// TIA Portal V15 export
// export: Created 2018-05-29T12:25:38.1552518Z, ExportSetting WithDefaults, DisplayName Totally Integrated Automation Portal, DisplayVersion V15, DisplayName TIA Portal Openness, DisplayVersion V15, DisplayName STEP 7 Professional, DisplayVersion V15, DisplayName WinCC Professional, DisplayVersion V15
FUNCTION "Control_Modules" : Void   // FC1, STL
TITLE = Program
{ S7_Optimized_Access := 'TRUE' }
VERSION : 0.1
// Call all the Control Modules
// stored: AutoNumber true, UDAEnableTagReadback false
BEGIN

NETWORK
TITLE = Main
// comment
	CALL	XV001_fc
	CALL	XV002_fc
	CALL	XV003_fc
	CALL	XV004_fc
	CALL	XV300_fc
	CALL	XV400_fc
	CALL	XV500_fc
	CALL	XV301_fc
	CALL	XV501_fc
	CALL	XV401_fc
	CALL	MV001_fc
	CALL	MV002_fc
	CALL	MV003_fc
	CALL	MV004_fc
	CALL	MV005_fc
	CALL	MV006_fc
	CALL	MV007_fc
	CALL	P100_fc
	CALL	P200_fc
	CALL	P101_fc
	CALL	P201_fc
	CALL	M100_fc
	CALL	M101_fc
	CALL	M102_fc
	CALL	M103_fc
	CALL	M104_fc
	CALL	M105_fc
	CALL	M106_fc
	CALL	LT001_fc
	CALL	LT002_fc
	CALL	LT003_fc
	CALL	LT004_fc
	CALL	LT005_fc
	CALL	LT006_fc
	CALL	LT007_fc
	CALL	LT100_fc
	CALL	LT200_fc
	CALL	LT101_fc
	CALL	LT201_fc
	CALL	LS001_fc
	CALL	LS002_fc
	CALL	LIC001_fc
	CALL	LIC002_fc
	CALL	LIC003_fc
	CALL	LIC004_fc
	CALL	LIC005_fc
	CALL	LIC006_fc
	CALL	FIC100_fc
	CALL	FIC101_fc
END_FUNCTION
